// TIA Portal V17 export
// export: Created 2022-07-20T07:02:39.6516597Z, ExportSetting WithDefaults, DisplayName Totally Integrated Automation Portal, DisplayVersion V17, DisplayName TIA Portal Openness, DisplayVersion V17, DisplayName TIA Portal Version Control Interface, DisplayVersion V17, DisplayName SINAMICS Startdrive Advanced, DisplayVersion V17, DisplayName SINAMICS Startdrive G130, G150, S120, S150, SINAMICS MV, S210, DisplayVersion V17, DisplayName SINAMICS Startdrive G110M, G120, G120C, G120D, G120P, G115D, DisplayVersion V17, DisplayName STEP 7 Professional, DisplayVersion V17, DisplayName STEP 7 Safety, DisplayVersion V17, DisplayName WinCC Advanced, DisplayVersion V17
VAR_GLOBAL   // PLC tag table "LCamHdl_AdditionalConstants"
END_VAR
VAR_GLOBAL CONSTANT   // user constants
   LCAMHDL_SINE_MODE_PHASE_START_AND_END : DInt := 0;
   LCAMHDL_SINE_MODE_PHASE_START_AND_PERIOD_LENGTH : DInt := 1;
   LCAMHDL_SINE_MODE_PHASE_START_AND_FREQUENCY : DInt := 2;
   LCAMHDL_SINE_MODE_PERIOD_LENGTH_AND_PHASE_END : DInt := 3;
   LCAMHDL_SINE_MODE_FREQUENCY_AND_PHASE_END : DInt := 4;
   LCAMHDL_SINE_INCL_MODE_DISPLACEMENT_START_AND_END : DInt := 0;
   LCAMHDL_SINE_INCL_MODE_DISPLACEMENT_START_AND_INCLINATION : DInt := 1;
   LCAMHDL_SINE_INCL_MODE_INCLINATION_AND_DISPLACEMENT_END : DInt := 2;
   LCAMHDL_POLY_MODE_BOUNDARY_VALUES_AND_POINT_OF_INFLECTION : DInt := 0;
   LCAMHDL_POLY_MODE_BOUNDARY_VALUES_AND_START_JERK : DInt := 1;
   LCAMHDL_POLY_MODE_BOUNDARY_VALUES_AND_END_JERK : DInt := 2;
END_VAR
